FUNCTION_BLOCK FB_LimSwStatus IMPLEMENTS I_LimSwStatus
VAR_INPUT
END_VAR
VAR_OUTPUT
END_VAR
VAR
    (* Hardware *)
   // NC Forward Limit Switch: TRUE if ok to move
    bLimitForwardEnable AT %I*: BOOL;
    // NC Backward Limit Switch: TRUE if ok to move
    bLimitBackwardEnable AT %I*: BOOL;
    // NO Home Switch: TRUE if at home
    bHome AT %I*: BOOL;

END_VAR

PROPERTY LimBackward : BOOL
GET
LimBackward := bLimitBackwardEnable;
END_GET
END_PROPERTY

PROPERTY LimForward : BOOL
GET
LimForward := bLimitForwardEnable;
END_GET
END_PROPERTY

PROPERTY LimHome : BOOL
GET
LimHome :=  bHome ;
END_GET
END_PROPERTY

PROPERTY MoveBackwardEnabled : BOOL
GET
MoveBackwardEnabled := bLimitBackwardEnable;
END_GET
END_PROPERTY

PROPERTY MoveForwardEnabled : BOOL
GET
MoveForwardEnabled :=  bLimitForwardEnable;
END_GET
END_PROPERTY

END_FUNCTION_BLOCK

(* stored: Version 1.1.0.1
   POU FB_LimSwStatus: Id {322e8186-deb9-4a53-b303-d1d3662306db}, SpecialFunc None
   Property LimBackward: Id {35aa245a-d874-4916-85c5-42c60fad40f0}
   Get Get: Id {5fbf77a3-1565-4123-a7e4-8abd4560ecb2}
   Property LimForward: Id {60bb8d48-4b37-425b-923e-b1e7d0d2cba8}
   Get Get: Id {c6fce77e-af19-46cd-b898-ad9a07ade412}
   Property LimHome: Id {1b597d59-cd48-4a23-82a2-a38399b4eb9e}
   Get Get: Id {a5e85be1-90e3-408d-830c-f40a8296404c}
   Property MoveBackwardEnabled: Id {89adc283-9c17-45ca-8f36-46140fc4dc4c}
   Get Get: Id {3db33672-1b0d-4c45-b399-57143d800f06}
   Property MoveForwardEnabled: Id {5cf35d17-2e51-4927-83dd-9d0c0496a7d4}
   Get Get: Id {157158b2-9f48-4b44-a9b9-77a750c8b408} *)
